SUBAPPLICATION Ventilsteuerung_Uebung_010b3 (* Toggle Flip-Flop mit IE AuxFunction2_X1 *)
  (* Standard: 61499-2 *)
  (* Version 1.0, 2023-10-23, franz *)
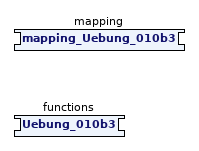
  SUBAPPS
    mapping : mapping_Uebung_010b3;
    functions : Uebung_010b3;
  END_SUBAPPS
END_SUBAPPLICATION
